AssertEquals(Expected := nExpectedState,
             Actual := nActualState,
             Message := 'State is not correct');	 
TEST_FINISHED();

TEST('Transition S3>S1_2');
fbDS402.eState := E_DS402State.S3_SwitchedOn;
fbDS402.stControl := GetQuickStopCommand();
fbDS402.stControl.b1_EnableVoltage := TRUE;
fbDS402();

nExpectedState := E_DS402State.S1_SwitchOnDisabled;
nActualState := fbDS402.eState;

AssertEquals(Expected := nExpectedState,
             Actual := nActualState,
             Message := 'State is not correct');	 
TEST_FINISHED();

TEST('Transition S3>S2');
fbDS402.eState := E_DS402State.S3_SwitchedOn;
fbDS402.stControl := GetShotdownCommand();
fbDS402();

nExpectedState := E_DS402State.S2_ReadyToSwitchOn;
nActualState := fbDS402.eState;

AssertEquals(Expected := nExpectedState,
             Actual := nActualState,
             Message := 'State is not correct');	 
TEST_FINISHED();

TEST('Transition S3>S4');
fbDS402.eState := E_DS402State.S3_SwitchedOn;
fbDS402.stControl := GetEnableCommand();
fbDS402();

nExpectedState := E_DS402State.S4_OperationEnabled;
nActualState := fbDS402.eState;

AssertEquals(Expected := nExpectedState,
             Actual := nActualState,
             Message := 'State is not correct');	 
TEST_FINISHED();
END_METHOD

METHOD TestState_S4 : BOOL
VAR
	fbDS402 			: FB_DS402FSM;
	stExpectedStatus 	: ST_DS402_6041h_StatusWord; 
	nMask 				: WORD;
	nResult 			: WORD;
	bResult 			: BOOL;
	nActualState		: INT;
	nExpectedState		: INT;
END_VAR
TEST('Set State S4');
fbDS402.eState := E_DS402State.S4_OperationEnabled;
fbDS402();

stExpectedStatus.b0_ReadyToSwitchOn 		:= TRUE;
stExpectedStatus.b1_SwitchedOn 				:= TRUE;
stExpectedStatus.b2_OperationEnabled		:= TRUE;
stExpectedStatus.b3_Fault					:= FALSE;
stExpectedStatus.b5_QuickStop 				:= TRUE; 
stExpectedStatus.b6_SwitchOnDisabled 		:= FALSE;

MEMCPY(ADR(nMask), ADR(stExpectedStatus), 2);
nResult := (2#01101111 AND fbDS402.nStatus);

AssertEquals(Expected := nMask,
             Actual := nResult,
             Message := 'Value is not correct');	 
TEST_FINISHED();

TEST('Transition S4>S6');
fbDS402.eState := E_DS402State.S4_OperationEnabled;
fbDS402.bError := TRUE;
fbDS402();
fbDS402.bError := FALSE;

nExpectedState := E_DS402State.S6_FaultReactionActive;
nActualState := fbDS402.eState;

AssertEquals(Expected := nExpectedState,
             Actual := nActualState,
             Message := 'State is not correct');	 
TEST_FINISHED();

TEST('Transition S4>S1');
fbDS402.eState := E_DS402State.S4_OperationEnabled;
fbDS402.stControl := GetDisableVoltageCommand();
fbDS402();

nExpectedState := E_DS402State.S1_SwitchOnDisabled;
nActualState := fbDS402.eState;

AssertEquals(Expected := nExpectedState,
             Actual := nActualState,
             Message := 'State is not correct');	 
TEST_FINISHED();

TEST('Transition S4>S2');
fbDS402.eState := E_DS402State.S4_OperationEnabled;
fbDS402.stControl := GetShotdownCommand();
fbDS402();

nExpectedState := E_DS402State.S2_ReadyToSwitchOn;
nActualState := fbDS402.eState;

AssertEquals(Expected := nExpectedState,
             Actual := nActualState,
             Message := 'State is not correct');	 
TEST_FINISHED();

TEST('Transition S4>S3');
fbDS402.eState := E_DS402State.S4_OperationEnabled;
fbDS402.stControl := GetDisableCommand();
fbDS402();

nExpectedState := E_DS402State.S3_SwitchedOn;
nActualState := fbDS402.eState;

AssertEquals(Expected := nExpectedState,
             Actual := nActualState,
             Message := 'State is not correct');	 
TEST_FINISHED();

TEST('Transition S4>S7');
fbDS402.eState := E_DS402State.S4_OperationEnabled;
fbDS402.stControl := GetQuickStopCommand();
fbDS402.stControl.b1_EnableVoltage := TRUE;
fbDS402();

nExpectedState := E_DS402State.S7_QuickStopActive;
nActualState := fbDS402.eState;

AssertEquals(Expected := nExpectedState,
             Actual := nActualState,
             Message := 'State is not correct');	 
TEST_FINISHED();
END_METHOD

METHOD TestState_S5 : BOOL
VAR
	fbDS402 			: FB_DS402FSM;
	stExpectedStatus 	: ST_DS402_6041h_StatusWord; 
	nMask 				: WORD;
	nResult 			: WORD;
	bResult 			: BOOL;
	nActualState		: INT;
	nExpectedState		: INT;
END_VAR
TEST('Set State S5');
fbDS402.eState := E_DS402State.S5_Fault;
fbDS402();

stExpectedStatus.b0_ReadyToSwitchOn 		:= FALSE;
stExpectedStatus.b1_SwitchedOn 				:= FALSE;
stExpectedStatus.b2_OperationEnabled		:= FALSE;
stExpectedStatus.b3_Fault					:= TRUE;
stExpectedStatus.b6_SwitchOnDisabled 		:= FALSE;

MEMCPY(ADR(nMask), ADR(stExpectedStatus), 2);
nResult := (2#01001111 AND fbDS402.nStatus);

AssertEquals(Expected := nMask,
             Actual := nResult,
             Message := 'Value is not correct');	 
TEST_FINISHED();

TEST('Transition S5>S1');
fbDS402.eState := E_DS402State.S5_Fault;
fbDS402.stControl.b7_FaultReset := TRUE;
fbDS402();
fbDS402.stControl.b7_FaultReset := FALSE;

nExpectedState := E_DS402State.S1_SwitchOnDisabled;
nActualState := fbDS402.eState;

AssertEquals(Expected := nExpectedState,
             Actual := nActualState,
             Message := 'State is not correct');	 
TEST_FINISHED();
END_METHOD

METHOD TestState_S6 : BOOL
VAR
	fbDS402 			: FB_DS402FSM;
	stExpectedStatus 	: ST_DS402_6041h_StatusWord; 
	nMask 				: WORD;
	nResult 			: WORD;
	bResult 			: BOOL;
	nActualState		: INT;
	nExpectedState		: INT;
END_VAR
TEST('Set State S6');
fbDS402.eState := E_DS402State.S6_FaultReactionActive;
fbDS402();

stExpectedStatus.b0_ReadyToSwitchOn 		:= TRUE;
stExpectedStatus.b1_SwitchedOn 				:= TRUE;
stExpectedStatus.b2_OperationEnabled		:= TRUE;
stExpectedStatus.b3_Fault					:= TRUE;
stExpectedStatus.b6_SwitchOnDisabled 		:= FALSE;

MEMCPY(ADR(nMask), ADR(stExpectedStatus), 2);
nResult := (2#01001111 AND fbDS402.nStatus);

AssertEquals(Expected := nMask,
             Actual := nResult,
             Message := 'Value is not correct');	 
TEST_FINISHED();

TEST('Transition S6>S5');
fbDS402.eState := E_DS402State.S6_FaultReactionActive;
fbDS402();

nExpectedState := E_DS402State.S5_Fault;
nActualState := fbDS402.eState;

AssertEquals(Expected := nExpectedState,
             Actual := nActualState,
             Message := 'State is not correct');	 
TEST_FINISHED();
END_METHOD

METHOD TestState_S7 : BOOL
VAR
	fbDS402 			: FB_DS402FSM;
	stExpectedStatus 	: ST_DS402_6041h_StatusWord; 
	nMask 				: WORD;
	nResult 			: WORD;
	bResult 			: BOOL;
	nActualState		: INT;
	nExpectedState		: INT;
END_VAR
TEST('Set State S7');
fbDS402.eState := E_DS402State.S7_QuickStopActive;
fbDS402();

stExpectedStatus.b0_ReadyToSwitchOn 		:= TRUE;
stExpectedStatus.b1_SwitchedOn 				:= TRUE;
stExpectedStatus.b2_OperationEnabled		:= TRUE;
stExpectedStatus.b3_Fault					:= FALSE;
stExpectedStatus.b5_QuickStop				:= FALSE;
stExpectedStatus.b6_SwitchOnDisabled 		:= FALSE;

MEMCPY(ADR(nMask), ADR(stExpectedStatus), 2);
nResult := (2#01101111 AND fbDS402.nStatus);

AssertEquals(Expected := nMask,
             Actual := nResult,
             Message := 'Value is not correct');	 
TEST_FINISHED();

TEST('Transition S7>S1');
fbDS402.eState := E_DS402State.S7_QuickStopActive;
fbDS402.stControl := GetDisableVoltageCommand();
fbDS402();

nExpectedState := E_DS402State.S1_SwitchOnDisabled;
nActualState := fbDS402.eState;

AssertEquals(Expected := nExpectedState,
             Actual := nActualState,
             Message := 'State is not correct');	 
TEST_FINISHED();

TEST('Transition S7>S4');
fbDS402.eState := E_DS402State.S7_QuickStopActive;
fbDS402.stControl := GetEnableCommand();
fbDS402();

nExpectedState := E_DS402State.S4_OperationEnabled;
nActualState := fbDS402.eState;

AssertEquals(Expected := nExpectedState,
             Actual := nActualState,
             Message := 'State is not correct');	 
TEST_FINISHED();
END_METHOD

END_FUNCTION_BLOCK

// Tests/Drives/FB_Encoder_Test
FUNCTION_BLOCK FB_Encoder_Test EXTENDS FB_TestSuite
VAR	
	stConfig 			: ST_EncoderConfig;
END_VAR

TestCase_Encoder('Absolute 1', 0, 0, LREAL_TO_DINT(0*1E4), stConfig);
TestCase_Encoder('Absolute 2', 100, 100, LREAL_TO_DINT(100*1E4), stConfig);
TestCase_Encoder('Absolute 3', -100, -100, LREAL_TO_DINT(-100*1E4), stConfig);

stConfig.fInputFactor := -1;
TestCase_Encoder('Absolute with Factor 1', 0, 0, LREAL_TO_DINT(0*1E4), stConfig);
TestCase_Encoder('Absolute with Factor 2', 100, -100, LREAL_TO_DINT(-100*1E4), stConfig);
TestCase_Encoder('Absolute with Factor 3', -100, 100, LREAL_TO_DINT(100*1E4), stConfig);

stConfig.fInputFactor := 1;
stConfig.bInvertIncrementValue := TRUE;
TestCase_Encoder('Absolute with Invert 1', 0, 0, LREAL_TO_DINT(0*1E4), stConfig);
TestCase_Encoder('Absolute with Invert 2', 100, 100, LREAL_TO_DINT(-100*1E4), stConfig);
TestCase_Encoder('Absolute with Invert 3', -100, -100, LREAL_TO_DINT(100*1E4), stConfig);

stConfig.fModulo := 360;
stConfig.bInvertIncrementValue := FALSE;
TestCase_Encoder('Modulo 1', 0, 0, LREAL_TO_DINT(0*1E4), stConfig);
TestCase_Encoder('Modulo 2', 360, 0, LREAL_TO_DINT(0*1E4), stConfig);
TestCase_Encoder('Modulo 3', 350, 350, LREAL_TO_DINT(350*1E4), stConfig);
TestCase_Encoder('Modulo 4', -350, -350, LREAL_TO_DINT(-350*1E4), stConfig);
TestCase_Encoder('Modulo 5', -360, 0, LREAL_TO_DINT(0*1E4), stConfig);

stConfig.fModulo := 0;
stConfig.bInvertIncrementValue := FALSE;
stConfig.bIsIntegral := TRUE;
TestCase_Encoder('Integrate 1', 0, 0, 0, stConfig);
TestCase_Encoder('Integrate 2', 100, 1, LREAL_TO_DINT(1*1E4), stConfig);
TestCase_Encoder('Integrate 3', -100, -1, LREAL_TO_DINT(-1*1E4), stConfig);

METHOD TestCase_Encoder
VAR_INPUT
	sName 					: T_MaxString;
	fInput					: REAL;
	fExpected				: LREAL;
	nExpected				: DINT;
	stConfig				: ST_EncoderConfig;
END_VAR

VAR	
	fbEncoder 				: FB_Encoder;
	nCycleCount 			: INT;
	fActual					: LREAL;	
	nActual					: DINT;	
	bValid 					: BOOL;
	fTolerance 				: REAL := 1E-6;
END_VAR
TEST(sName);

fbEncoder.stConfig := stConfig;
fbEncoder.fInput := fInput;

(*	Call FB to test	*)
FOR nCycleCount := 0 TO 9 DO
   fbEncoder();
END_FOR

(*	Evaluation of results	*)
nActual := fbEncoder.nPosition;
fActual := fbEncoder.fPosition;

AssertEquals(Expected := nExpected,
             Actual := nActual,
             Message := 'nPosition is not correct');

bValid := ABS(fExpected - fActual) < fTolerance;			 
	
AssertTrue(bValid, 'fPosition is not correct');

TEST_FINISHED();
END_METHOD

END_FUNCTION_BLOCK

// Tests/Drives/FB_SimMovidriveFSM_Test
FUNCTION_BLOCK FB_SimMovidriveFSM_Test EXTENDS TcUnit.FB_TestSuite

// TestState(sTestInfo, bControllerInhibit, bRapidStop,	bStop,	bHoldControl, eInitState, eExpectedState)	

// ControllerInhibit
TestState('ControllerInhibit, no transition', TRUE, FALSE, FALSE, FALSE, E_SimMovitracState.ControllerInhibit, E_SimMovitracState.ControllerInhibit);
TestState('ControllerInhibit -> RapidStop', FALSE, FALSE, FALSE, FALSE, E_SimMovitracState.ControllerInhibit, E_SimMovitracState.RapidStop);

//  RapidStop 
TestState('RapidStop, no transition', FALSE, FALSE, FALSE, FALSE, E_SimMovitracState.RapidStop, E_SimMovitracState.RapidStop);
TestState('RapidStop -> ControllerInhibit', TRUE, FALSE, FALSE, FALSE, E_SimMovitracState.RapidStop, E_SimMovitracState.ControllerInhibit);
TestState('RapidStop -> Halt', FALSE, TRUE, FALSE, FALSE, E_SimMovitracState.RapidStop, E_SimMovitracState.Halt);

// Halt
TestState('Halt, no transition', FALSE, TRUE, FALSE, FALSE, E_SimMovitracState.Halt, E_SimMovitracState.Halt);
TestState('Halt -> ControllerInhibit', TRUE, FALSE, FALSE, FALSE, E_SimMovitracState.Halt, E_SimMovitracState.ControllerInhibit);
TestState('Halt -> RapidStop', FALSE, FALSE, FALSE, FALSE, E_SimMovitracState.Halt, E_SimMovitracState.RapidStop);
TestState('Halt -> HoldControl', FALSE, TRUE, TRUE, TRUE, E_SimMovitracState.Halt, E_SimMovitracState.HoldControl);
TestState('Halt -> Enable', FALSE, TRUE, TRUE, FALSE, E_SimMovitracState.Halt, E_SimMovitracState.Enable);

// Enable
TestState('Enable, no transition', FALSE, TRUE, TRUE, FALSE, E_SimMovitracState.Enable, E_SimMovitracState.Enable);
TestState('Enable -> ControllerInhibit', TRUE, FALSE, FALSE, FALSE, E_SimMovitracState.Enable, E_SimMovitracState.ControllerInhibit);
TestState('Enable -> RapidStop', FALSE, FALSE, FALSE, FALSE, E_SimMovitracState.Enable, E_SimMovitracState.RapidStop);
TestState('Enable -> Halt', FALSE, TRUE, FALSE, FALSE, E_SimMovitracState.Enable, E_SimMovitracState.Halt);
TestState('Enable -> HoldControl', FALSE, TRUE, TRUE, TRUE, E_SimMovitracState.Enable, E_SimMovitracState.HoldControl);

// HoldControl
TestState('HoldControl, no transition', FALSE, TRUE, TRUE, TRUE, E_SimMovitracState.HoldControl, E_SimMovitracState.HoldControl);
TestState('HoldControl -> ControllerInhibit', TRUE, FALSE, FALSE, FALSE, E_SimMovitracState.HoldControl, E_SimMovitracState.ControllerInhibit);
TestState('HoldControl -> RapidStop', FALSE, FALSE, FALSE, FALSE, E_SimMovitracState.HoldControl, E_SimMovitracState.RapidStop);
TestState('HoldControl -> Halt', FALSE, TRUE, FALSE, FALSE, E_SimMovitracState.HoldControl, E_SimMovitracState.Halt);
TestState('HoldControl -> Enable', FALSE, TRUE, TRUE, FALSE, E_SimMovitracState.HoldControl, E_SimMovitracState.Enable);

METHOD TestState : BOOL
VAR_INPUT
	sTestInfo			: T_MaxString;
	bControllerInhibit	: BOOL;
	bRapidStop			: BOOL;
	bStop				: BOOL;
	bHoldControl		: BOOL;
	eInitState			: E_SimMovitracState;	
	eExpectedState		: E_SimMovitracState;	
END_VAR

VAR
		fbMovidriveStateMachine		: FB_SimMovitracFSM;
END_VAR
TEST(sTestInfo);

fbMovidriveStateMachine.bControllerInhibit := bControllerInhibit;
fbMovidriveStateMachine.bRapidStop := bRapidStop;
fbMovidriveStateMachine.bStop := bStop;
fbMovidriveStateMachine.bHoldControl := bHoldControl;

fbMovidriveStateMachine.nState := eInitState;

fbMovidriveStateMachine();

AssertEquals(Expected := eExpectedState,
             Actual := fbMovidriveStateMachine.eState,
             Message := 'State is not correct');
	 
TEST_FINISHED();
END_METHOD

END_FUNCTION_BLOCK

// Tests/Drives/FB_SimMovidrivePDO12_Test
FUNCTION_BLOCK FB_SimMovidrivePDO12_Test EXTENDS TcUnit.FB_TestSuite
VAR_INPUT
END_VAR
VAR_OUTPUT
END_VAR
VAR
END_VAR

Test_GetControlMode();
Test_GetControlData();
Test_GetControlDataSWAP();
Test_SetStatusData();
Test_SetStatusDataSWAP();

METHOD Test_AssignProcessData : REFERENCE TO FB_Test
VAR
	fbStarter 				: FB_Starter;
	nControlData 			: WORD;
	nStatusData				: WORD;
	
	nExpectedStatusData		: WORD;
	
	nActualControlData 		: WORD;
	nActualStatusData		: WORD;
	stActualControlData 	: ST_StarterControlData;
	stActualStatusData		: ST_StarterStatusData;
END_VAR
TEST('Assign Process data');

nControlData := 255;
nStatusData := 0;

fbStarter.AssignProcessData(nControlData, nStatusData);
fbStarter();

stActualControlData := fbStarter.stControlData;
stActualStatusData := fbStarter.stStatusData;

MEMCPY(ADR(nActualControlData), ADR(stActualControlData), 2);
MEMCPY(ADR(nActualStatusData), ADR(stActualStatusData), 2);

AssertEquals(Expected := nControlData,
             Actual := nActualControlData,
             Message := 'nControlData is not correct');	
		
nExpectedStatusData := 1;
	 
AssertEquals(Expected := nExpectedStatusData,
             Actual := nStatusData,
             Message := 'nStatusData is not correct');	

TEST_FINISHED();
END_METHOD

METHOD Test_GetControlData : BOOL
VAR
	stDataBus 		: ST_SimMovidriveControlData;
	stControl 		: ST_SimMovidriveControlData;
	stExpected 		: ST_SimMovidriveControlData;
	fbMoviPos_PD12 	: FB_SimMovidrivePDO12;
	
	nControlWord	: WORD;
	nControlWordExpected	: WORD;
END_VAR
TEST('Get Control Data');

stDataBus.bControllerInhibit := TRUE;
stDataBus.nTargetPosition := 100;
stDataBus.nVelocity := 200;
stDataBus.nAcceleration := 300;
stDataBus.nDeceleration := 400;

stExpected := stDataBus;
MEMCPY(ADR(nControlWordExpected), ADR(stExpected), 2);

fbMoviPos_PD12.GetControlData(stControl, ADR(stDataBus), FALSE);
MEMCPY(ADR(nControlWord), ADR(stControl), 2);

AssertEquals(Expected := nControlWordExpected,
             Actual := nControlWord,
             Message := 'nControlWord is not equal');
			 
AssertEquals(Expected := stExpected.nTargetPosition,
             Actual := stControl.nTargetPosition,
             Message := 'nTargetPosition word is not equal');
			 
AssertEquals(Expected := stExpected.nVelocity,
             Actual := stControl.nVelocity,
             Message := 'nVelocity word is not equal');	
			 
AssertEquals(Expected := stExpected.nAcceleration,
             Actual := stControl.nAcceleration,
             Message := 'nAcceleration word is not equal');	

AssertEquals(Expected := stExpected.nDeceleration,
             Actual := stControl.nDeceleration,
             Message := 'nAcceleration word is not equal');		 
		
TEST_FINISHED();
END_METHOD

METHOD Test_GetControlDataSWAP : BOOL
VAR
	stDataBus 				: ST_SimMovidriveControlData;
	stControl 				: ST_SimMovidriveControlData;
	stExpected 				: ST_SimMovidriveControlData;
	fbMoviPos_PD12 			: FB_SimMovidrivePDO12;
	                		
	nControlWord			: WORD;
	nControlWordExpected	: WORD;	
	nBusControlWord			: WORD;
END_VAR
TEST('Get Control Data SWAP');

nControlWordExpected := 15;
MEMCPY(ADR(stExpected), ADR(nControlWordExpected), 2);
stExpected.nTargetPosition := 100;
stExpected.nVelocity := 200;
stExpected.nAcceleration := 300;
stExpected.nDeceleration := 400;

stDataBus := stExpected ;
MEMCPY(ADR(nBusControlWord), ADR(stDataBus), 2);
nBusControlWord := HOST_TO_BE16(nBusControlWord);
MEMCPY(ADR(stDataBus), ADR(nBusControlWord), 2);

stDataBus.nTargetPosition := DWORD_TO_DINT(HOST_TO_BE32(DINT_TO_DWORD(stDataBus.nTargetPosition)));
stDataBus.nVelocity := HOST_TO_BE16(stDataBus.nVelocity);
stDataBus.nAcceleration := HOST_TO_BE16(stDataBus.nAcceleration);
stDataBus.nDeceleration := HOST_TO_BE16(stDataBus.nDeceleration);

fbMoviPos_PD12.GetControlData(stControl, ADR(stDataBus), TRUE);
MEMCPY(ADR(nControlWord), ADR(stControl), 2);

AssertEquals(Expected := nControlWordExpected,
             Actual := nControlWord,
             Message := 'nControlWord is not equal');
			 
AssertEquals(Expected := stExpected.nTargetPosition,
             Actual := stControl.nTargetPosition,
             Message := 'nTargetPosition word is not equal');
			 
AssertEquals(Expected := stExpected.nVelocity,
             Actual := stControl.nVelocity,
             Message := 'nVelocity word is not equal');	
			 
AssertEquals(Expected := stExpected.nAcceleration,
             Actual := stControl.nAcceleration,
             Message := 'nAcceleration word is not equal');	

AssertEquals(Expected := stExpected.nDeceleration,
             Actual := stControl.nDeceleration,
             Message := 'nAcceleration word is not equal');		 
		
TEST_FINISHED();
END_METHOD

METHOD Test_GetControlMode : REFERENCE TO FB_Test
VAR
	stControl 		: ST_SimMovidriveControlData;
	fbMoviPos_PD12 	: FB_SimMovidrivePDO12;
	bExpected		: BOOL;
	bResult			: BOOL;
END_VAR
TEST('Get Control Mode');

stControl.bModeLow := FALSE;
stControl.bModeHigh := FALSE;
bResult := fbMoviPos_PD12.GetControlMode(stControl) = E_SimMovidriveMode.Idle;
AssertTrue(bResult, 'Expected Idle Mode');


stControl.bModeLow := TRUE;
stControl.bModeHigh := FALSE;
bResult := fbMoviPos_PD12.GetControlMode(stControl) = E_SimMovidriveMode.Jog;
AssertTrue(bResult, 'Expected Jog Mode');

stControl.bModeLow := FALSE;
stControl.bModeHigh := TRUE;
bResult := fbMoviPos_PD12.GetControlMode(stControl) = E_SimMovidriveMode.Ref;
AssertTrue(bResult, 'Expected Ref Mode');

stControl.bModeLow := TRUE;
stControl.bModeHigh := TRUE;
bResult := fbMoviPos_PD12.GetControlMode(stControl) = E_SimMovidriveMode.Auto;
AssertTrue(bResult, 'Expected Auto Mode');

TEST_FINISHED();
END_METHOD

METHOD Test_SetStatusData : BOOL
VAR
	stControl 				: ST_SimMovidriveStatusData;
	stBuffer				: ST_SimMovidriveStatusData;
	fbMoviPos_PD12 			: FB_SimMovidrivePDO12;	                		
	nControlStatusByte		: BYTE;
	nActualStatusByte		: BYTE;
	nStatusWordSwap			: WORD;
END_VAR
TEST('Set Status Data');

nControlStatusByte := 124;
MEMCPY(ADR(stControl), ADR(nControlStatusByte), 1);
stControl.nStatus := 164;
stControl.nActPosition := 100;
stControl.nActVelocity := 200;
stControl.nActCurrent := 300;
stControl.nActUnit := 400;

fbMoviPos_PD12.SetStatusData(stControl, ADR(stBuffer), FALSE);

MEMCPY(ADR(nActualStatusByte), ADR(stBuffer), 1);

AssertEquals(Expected := nControlStatusByte,
             Actual := nActualStatusByte,
             Message := 'nExpectedStatusByte is not equal');

AssertEquals(Expected := stControl.nStatus,
             Actual := stBuffer.nStatus,
             Message := 'nStatus word is not equal');	

AssertEquals(Expected := stControl.nActPosition,
             Actual := stBuffer.nActPosition,
             Message := 'nActPosition word is not equal'); 
			 
AssertEquals(Expected := stControl.nActVelocity,
             Actual := stBuffer.nActVelocity,
             Message := 'nActVelocity word is not equal');
			 
AssertEquals(Expected := stControl.nActCurrent,
             Actual := stBuffer.nActCurrent,
             Message := 'nActCurrent word is not equal');
			 
AssertEquals(Expected := stControl.nActUnit,
             Actual := stBuffer.nActUnit,
             Message := 'nActCurrent word is not equal');

TEST_FINISHED();
END_METHOD

METHOD Test_SetStatusDataSWAP : BOOL
VAR
	stControl 				: ST_SimMovidriveStatusData;
	stBuffer				: ST_SimMovidriveStatusData;
	fbMoviPos_PD12 			: FB_SimMovidrivePDO12;	                		
	nControlStatusByte		: BYTE;
	nActualStatusByte		: BYTE;
	nStatusWordSwap			: WORD;
END_VAR
TEST('Set Status Data SWAP');

nControlStatusByte := 124;
MEMCPY(ADR(stControl), ADR(nControlStatusByte), 1);
stControl.nStatus := 164;
stControl.nActPosition := 100;
stControl.nActVelocity := 200;
stControl.nActCurrent := 300;
stControl.nActUnit := 400;

fbMoviPos_PD12.SetStatusData(stControl, ADR(stBuffer), TRUE);

MEMCPY(ADR(nStatusWordSwap), ADR(stBuffer), 2);
nStatusWordSwap := HOST_TO_BE16(nStatusWordSwap);
MEMCPY(ADR(stBuffer), ADR(nStatusWordSwap), 2);
stBuffer.nActPosition := DWORD_TO_DINT(HOST_TO_BE32(DINT_TO_DWORD(stBuffer.nActPosition)));
stBuffer.nActVelocity := HOST_TO_BE16(stBuffer.nActVelocity);
stBuffer.nActCurrent := HOST_TO_BE16(stBuffer.nActCurrent);
stBuffer.nActUnit := HOST_TO_BE16(stBuffer.nActUnit);

MEMCPY(ADR(nActualStatusByte), ADR(stBuffer), 1);

AssertEquals(Expected := nControlStatusByte,
             Actual := nActualStatusByte,
             Message := 'nExpectedStatusByte is not equal');

AssertEquals(Expected := stControl.nStatus,
             Actual := stBuffer.nStatus,
             Message := 'nStatus word is not equal');	

AssertEquals(Expected := stControl.nActPosition,
             Actual := stBuffer.nActPosition,
             Message := 'nActPosition word is not equal'); 
			 
AssertEquals(Expected := stControl.nActVelocity,
             Actual := stBuffer.nActVelocity,
             Message := 'nActVelocity word is not equal');
			 
AssertEquals(Expected := stControl.nActCurrent,
             Actual := stBuffer.nActCurrent,
             Message := 'nActCurrent word is not equal');
			 
AssertEquals(Expected := stControl.nActUnit,
             Actual := stBuffer.nActUnit,
             Message := 'nActUnit word is not equal');

TEST_FINISHED();
END_METHOD

END_FUNCTION_BLOCK

// Tests/Drives/FB_SimMovitrac_Test
FUNCTION_BLOCK FB_SimMovitrac_Test EXTENDS FB_TestSuite
VAR
	fbMovitrac : FB_SimMovitrac;
END_VAR

// No Movement
Test_Movitrac('No Movement, No STO', FALSE, FALSE, TRUE, TRUE, 1000, 0, FALSE, 10);
Test_Movitrac('No Movement, ControllerInhibit', TRUE, TRUE, TRUE, TRUE, 1000, 0, FALSE, 10);
Test_Movitrac('No Movement, No RapidStop', TRUE, FALSE, FALSE, TRUE, 1000, 0, FALSE, 10);
Test_Movitrac('No Movement, No Stop', TRUE, FALSE, TRUE, FALSE, 1000, 0, FALSE, 10);

// Movement
Test_Movitrac('Velocity postive', TRUE, FALSE, TRUE, TRUE, 1000, 1000, TRUE, 50);
Test_Movitrac('Velocity negative', TRUE, FALSE, TRUE, TRUE, -1000, -1000, TRUE, 50);
Test_Movitrac('Velocity 0', TRUE, FALSE, TRUE, TRUE, 0, 0, FALSE, 50);

// Stop
Test_Movitrac('Velocity to Stop', TRUE, FALSE, TRUE, TRUE, 1000, 1000, TRUE, 50);
Test_Movitrac('Stop', TRUE, FALSE, TRUE, FALSE, 0, 0, FALSE, 50);

// Rapid Stop
Test_Movitrac('Velocity to Rapid Stop', TRUE, FALSE, TRUE, TRUE, 1000, 1000, TRUE, 50);
Test_Movitrac('Rapid Stop', TRUE, FALSE, FALSE, TRUE, 0, 0, FALSE, 50);

// STO Stop
Test_Movitrac('Velocity to STO Stop', TRUE, FALSE, TRUE, TRUE, 1000, 1000, TRUE, 50);
Test_Movitrac('STO Stop', FALSE, FALSE, TRUE, TRUE, 0, 0, FALSE, 50);

METHOD Test_Movitrac
VAR
	nCycleCount : INT;
	bResultOutputStage : BOOL;
END_VAR
VAR_INPUT
	sTestInfo			: T_MaxString;
	bSto				: BOOL;
	bControllerInhibit	: BOOL;
	bRapidStop			: BOOL;
	bStop				: BOOL;
	nSetpointSpeed		: INT;	
	eExpectedSpeed		: INT;
	bExpectedOutputStage: BOOL;		
	bCycles				: INT;	
END_VAR
TEST(sTestInfo);

fbMovitrac.bSTO := bSTO;
fbMovitrac.stControlData.bControllerInhibit := bControllerInhibit;
fbMovitrac.stControlData.bRapidStop := bRapidStop;
fbMovitrac.stControlData.bStop := bStop;
fbMovitrac.stControlData.nSetpointSpeed := nSetpointSpeed; 

FOR nCycleCount := 0 TO bCycles DO
    fbMovitrac();
END_FOR

bResultOutputStage := fbMovitrac.stStatusData.bEnableOutputStage;

AssertEquals(Expected := eExpectedSpeed,
             Actual := fbMovitrac.stStatusData.nActSpeed,
             Message := 'Velocity/Speed is not correct');
			 
AssertEquals(Expected := bExpectedOutputStage,
             Actual := bResultOutputStage,
             Message := 'EnableOutputStage is not correct');

TEST_FINISHED();
END_METHOD

END_FUNCTION_BLOCK

// Tests/Drives/FB_SimMovitracB_Test
FUNCTION_BLOCK FB_SimMovitracB_Test EXTENDS FB_TestSuite
VAR
	fbMovitracB : FB_SimMovitracB;
END_VAR

// No Movement
TestCase_SimMovitracB('No Movement, No STO', FALSE, FALSE, TRUE, TRUE, 32767, 0, FALSE);
TestCase_SimMovitracB('No Movement, ControllerInhibit', TRUE, TRUE, TRUE, TRUE, 32767, 0, FALSE);
TestCase_SimMovitracB('No Movement, No RapidStop', TRUE, FALSE, FALSE, TRUE, 32767, 0, FALSE);
TestCase_SimMovitracB('No Movement, No Stop', TRUE, FALSE, TRUE, FALSE, 32767, 0, FALSE);

// Movement
TestCase_SimMovitracB('Velocity postive', TRUE, FALSE, TRUE, TRUE, 32767, 3000, TRUE);
TestCase_SimMovitracB('Velocity negative', TRUE, FALSE, TRUE, TRUE, -32767, -3000, TRUE);
TestCase_SimMovitracB('Velocity 0', TRUE, FALSE, TRUE, TRUE, 0, 0, FALSE);

// Stop
TestCase_SimMovitracB('Velocity to Stop', TRUE, FALSE, TRUE, TRUE, 32767, 3000, TRUE);
TestCase_SimMovitracB('Stop', TRUE, FALSE, TRUE, FALSE, 0, 0, FALSE);

// STO Stop
TestCase_SimMovitracB('Velocity to STO Stop', TRUE, FALSE, TRUE, TRUE, 32767, 3000, TRUE);
TestCase_SimMovitracB('STO Stop', FALSE, FALSE, TRUE, TRUE, 0, 0, FALSE);

// Rapid Stop
TestCase_SimMovitracB('Velocity to Rapid Stop', TRUE, FALSE, TRUE, TRUE, 32767, 3000, TRUE);
TestCase_SimMovitracB('Rapid Stop', TRUE, FALSE, FALSE, TRUE, 0, 0, FALSE);

METHOD TestCase_SimMovitracB
VAR
	nCycleCount : INT;
	bResultOutputStage : BOOL;
END_VAR
VAR_INPUT
	sTestInfo			: T_MaxString;
	bSto				: BOOL;
	bControllerInhibit	: BOOL;
	bRapidStop			: BOOL;
	bStop				: BOOL;
	nSetpointSpeed		: INT;	
	eExpectedSpeed		: REAL;
	bExpectedOutputStage: BOOL;		
END_VAR
TEST(sTestInfo);

fbMovitracB.bSTO := bSTO;
fbMovitracB.stControlData.bControllerInhibit := bControllerInhibit;
fbMovitracB.stControlData.bRapidStop := bRapidStop;
fbMovitracB.stControlData.bStop := bStop;
fbMovitracB.stControlData.nSetpointSpeed := nSetpointSpeed; 

fbMovitracB();

bResultOutputStage := fbMovitracB.stStatusData.bEnableOutputStage;

AssertEquals(Expected := eExpectedSpeed,
             Actual := fbMovitracB.fVelocity,
             Message := 'Velocity/Speed is not correct');
			 
AssertEquals(Expected := bExpectedOutputStage,
             Actual := bResultOutputStage,
             Message := 'EnableOutputStage is not correct');

TEST_FINISHED();
END_METHOD

END_FUNCTION_BLOCK

// Tests/Drives/FB_SimMovitracLTEB_Test
FUNCTION_BLOCK FB_SimMovitracLTEB_Test EXTENDS FB_TestSuite
VAR
	fbMovitracLTE : FB_SimMovitracLTEB;
	nExpectedByte : BYTE;
	nResultByte : BYTE;
	fExpectedReal : REAL;
	fResultReal : REAL;
	bExpectedBool : BOOL;
	bResultBool : BOOL;
END_VAR

Test_DriveNotReady();
Test_DriveReady();
Test_DriveRunningFwd();
Test_DriveRunningBwd();

METHOD Test_DriveNotReady
VAR_INPUT
END_VAR
TEST('Drive is not ready');
nExpectedByte := 0; 
bExpectedBool := FALSE;
fbMovitracLTE.bEnable := FALSE;
fbMovitracLTE.bSTO := FALSE;
fbMovitracLTE();
nResultByte := fbMovitracLTE.GetControl();
bResultBool := fbMovitracLTE.bReady;
AssertEquals(Expected := nExpectedByte,
             Actual := nResultByte,
             Message := 'Value is not correct');

AssertEquals(Expected := bExpectedBool, 
			 Actual := bResultBool,
			 Message := 'Status is not correct');	
TEST_FINISHED();
END_METHOD

METHOD Test_DriveReady
VAR_INPUT
END_VAR
TEST('Drive is ready');
nExpectedByte := 0; 
bExpectedBool := TRUE;
fbMovitracLTE.bEnable := FALSE;
fbMovitracLTE.bSTO := TRUE;
fbMovitracLTE();
nResultByte := fbMovitracLTE.GetControl();
bResultBool := fbMovitracLTE.bReady;

AssertEquals(Expected := nExpectedByte,
             Actual := nResultByte,
             Message := 'Value is not correct');

AssertEquals(Expected := bExpectedBool,
			 Actual := bResultBool,
			 Message := 'Status is not correct');	
TEST_FINISHED();
END_METHOD

METHOD Test_DriveRunningBwd
VAR_INPUT
END_VAR
TEST('Drive is running backward with 0 speed');
fbMovitracLTE.bSTO := TRUE;
fbMovitracLTE.bReverse := TRUE;
fExpectedReal := 0;
bExpectedBool := TRUE;
fbMovitracLTE.bEnable := TRUE;
fbMovitracLTE.nTargetSpeed := 0;
fbMovitracLTE.SetStatus(1);
fbMovitracLTE();
fResultReal := fbMovitracLTE.GetLinkControlData();
bResultBool := fbMovitracLTE.bRunning;

AssertEquals(Expected := fExpectedReal,
             Actual := fResultReal,
             Message := 'DataOut is not correct');	
			 
AssertEquals(Expected := bExpectedBool,
             Actual := bResultBool,
             Message := 'Status is not correct');	
			 
TEST_FINISHED();
//######################################################
TEST('Feedback of Drive running backward with 0 speed');
fbMovitracLTE.bSTO := TRUE;
fbMovitracLTE.bReverse := TRUE;
fExpectedReal := 0;
bExpectedBool := TRUE;
fbMovitracLTE.bEnable := TRUE;
fbMovitracLTE.nTargetSpeed := 0;
fbMovitracLTE.SetLinkStatusData(fExpectedReal);
fbMovitracLTE.SetStatus(1);
fbMovitracLTE();
fResultReal := fbMovitracLTE.fActualSpeed;
bResultBool := fbMovitracLTE.bRunning;

AssertEquals(Expected := fExpectedReal,
             Actual := fResultReal,
             Message := 'DataIn is not correct');	
			 
AssertEquals(Expected := bExpectedBool,
             Actual := bResultBool,
             Message := 'Status is not correct');	
			 
TEST_FINISHED();
//######################################################
TEST('Drive is running backward at max speed');
fbMovitracLTE.bSTO := TRUE;
fbMovitracLTE.bReverse := TRUE;
fExpectedReal := -3000.0;
bExpectedBool := TRUE;
fbMovitracLTE.bEnable := TRUE;
fbMovitracLTE.nTargetSpeed := 65535;
fbMovitracLTE.SetStatus(1);
fbMovitracLTE();
fResultReal := fbMovitracLTE.GetLinkControlData();
bResultBool := fbMovitracLTE.bRunning;

AssertEquals(Expected := fExpectedReal,
             Actual := fResultReal,
             Message := 'DataOut is not correct');	
			 
AssertEquals(Expected := bExpectedBool,
             Actual := bResultBool,
             Message := 'Status is not correct');	
			 
TEST_FINISHED();
//###################################################
TEST('Feedback of Drive running backward at max speed');
fbMovitracLTE.bSTO := TRUE;
fbMovitracLTE.bReverse := TRUE;
fExpectedReal := 0;
bExpectedBool := TRUE;
fbMovitracLTE.bEnable := TRUE;
fbMovitracLTE.nTargetSpeed := 0;
fbMovitracLTE.SetStatus(1);
fbMovitracLTE.SetLinkStatusData(fExpectedReal);
fbMovitracLTE();
fResultReal := fbMovitracLTE.fActualSpeed;
bResultBool := fbMovitracLTE.bRunning;

AssertEquals(Expected := fExpectedReal,
             Actual := fResultReal,
             Message := 'DataIn is not correct');	
			 
AssertEquals(Expected := bExpectedBool,
             Actual := bResultBool,
             Message := 'Status is not correct');	
			 
TEST_FINISHED();
END_METHOD

METHOD Test_DriveRunningFwd
VAR_INPUT
END_VAR
TEST('Drive is running forward at 0');
fExpectedReal := 0;
bExpectedBool := TRUE;
fbMovitracLTE.bSTO := TRUE;
fbMovitracLTE.nTargetSpeed := 0;
fbMovitracLTE.bEnable := TRUE;
fbMovitracLTE.SetStatus(1);
fbMovitracLTE();
fResultReal := fbMovitracLTE.GetLinkControlData();
bResultBool := fbMovitracLTE.bRunning;

AssertEquals(Expected := fExpectedReal,
             Actual := fResultReal,
             Message := 'DataOut is not correct');	

AssertEquals(Expected := bExpectedBool, 
			 Actual := bResultBool,
			 Message := 'Status is not correct');
TEST_FINISHED();
//#################################################################
TEST('Feedback of drive running forward at 0');
fExpectedReal := 0;
bExpectedBool := TRUE;
fbMovitracLTE.bSTO := TRUE;
fbMovitracLTE.nTargetSpeed := 0;
fbMovitracLTE.bEnable := TRUE;
fbMovitracLTE.SetStatus(1);
fbMovitracLTE.SetLinkStatusData(fExpectedReal);
fbMovitracLTE();
fResultReal := fbMovitracLTE.fActualSpeed;
bResultBool := fbMovitracLTE.bRunning;

AssertEquals(Expected := fExpectedReal,
             Actual := fResultReal,
             Message := 'DataIn is not correct');	

AssertEquals(Expected := bExpectedBool, 
			 Actual := bResultBool,
			 Message := 'Status is not correct');
TEST_FINISHED();
//###################################################################
TEST('Drive is running forward at max speed');
fExpectedReal := 3000;
bExpectedBool := TRUE;
fbMovitracLTE.bSTO := TRUE;
fbMovitracLTE.nTargetSpeed := 65535;
fbMovitracLTE.bEnable := TRUE;
fbMovitracLTE.SetStatus(1);
fbMovitracLTE();
fResultReal := fbMovitracLTE.GetLinkControlData();
bResultBool := fbMovitracLTE.bRunning;

AssertEquals(Expected := fExpectedReal,
             Actual := fResultReal,
             Message := 'DataOut is not correct');	

AssertEquals(Expected := bExpectedBool, 
			 Actual := bResultBool,
			 Message := 'Status is not correct');
TEST_FINISHED();
//###################################################################
TEST('Feedback of drive running forward at max speed');
fExpectedReal := 3000;
bExpectedBool := TRUE;
fbMovitracLTE.bSTO := TRUE;
fbMovitracLTE.nTargetSpeed := 65535;
fbMovitracLTE.bEnable := TRUE;
fbMovitracLTE.SetStatus(1);
fbMovitracLTE.SetLinkStatusData(fExpectedReal);
fbMovitracLTE();
fResultReal := fbMovitracLTE.fActualSpeed;
bResultBool := fbMovitracLTE.bRunning;

AssertEquals(Expected := fExpectedReal,
             Actual := fResultReal,
             Message := 'DataIn is not correct');	

AssertEquals(Expected := bExpectedBool, 
			 Actual := bResultBool,
			 Message := 'Status is not correct');
TEST_FINISHED();
END_METHOD

END_FUNCTION_BLOCK

// Tests/Drives/FB_Starter_Test
FUNCTION_BLOCK FB_Starter_Test EXTENDS FB_TestSuite
VAR
	fbStarter : FB_Starter;
	
	fExpectedReal 		: REAL;
	fResultReal 		: REAL;
	bExpectedBool 		: BOOL;
	bResultBool 		: BOOL;
	fExpectedDataOut 	: REAL;
END_VAR

Test_GetControlData();
Test_GetControlDataSWAP();
Test_SetStatusData();
Test_SetStatusDataSWAP();

//Test_DriveNoMovement();
//Test_DriveRunningCw();
//Test_DriveRunningCcw();
//Test_AssignProcessData();

METHOD Test_AssignProcessData : REFERENCE TO FB_Test
VAR
	fbStarter 				: FB_Starter;
	nControlData 			: WORD;
	nStatusData				: WORD;
	
	nExpectedStatusData		: WORD;
	
	nActualControlData 		: WORD;
	nActualStatusData		: WORD;
	stActualControlData 	: ST_StarterControlData;
	stActualStatusData		: ST_StarterStatusData;
END_VAR
TEST('Assign Process data');

nControlData := 255;
nStatusData := 0;

fbStarter.AssignProcessData(nControlData, nStatusData);
fbStarter();

stActualControlData := fbStarter.stControlData;
stActualStatusData := fbStarter.stStatusData;

MEMCPY(ADR(nActualControlData), ADR(stActualControlData), 2);
MEMCPY(ADR(nActualStatusData), ADR(stActualStatusData), 2);

AssertEquals(Expected := nControlData,
             Actual := nActualControlData,
             Message := 'nControlData is not correct');	
		
nExpectedStatusData := 1;
	 
AssertEquals(Expected := nExpectedStatusData,
             Actual := nStatusData,
             Message := 'nStatusData is not correct');	

TEST_FINISHED();
END_METHOD

METHOD Test_DriveNoMovement
VAR
	nCycleCount : INT;	
END_VAR
TEST('Starter no movement, CW/CCW missing');

fbStarter.stConfig.fVelocity := 10;
fbStarter.stConfig.fAcceleration := 1000;
fbStarter.stConfig.fDeceleration := 1000;

fbStarter.stControlData.MotorCW := FALSE;
fbStarter.stControlData.MotorCCW := FALSE;
fbStarter.stControlData.BrakeActuation := TRUE;

fExpectedReal := 0;
bExpectedBool := FALSE;

FOR nCycleCount := 0 TO 10 DO
    fbStarter();
END_FOR

fResultReal := fbStarter.fSpeed;
bResultBool := fbStarter.stStatusData.MotorON;

AssertEquals(Expected := fExpectedReal,
             Actual := fResultReal,
             Message := 'fSpeed is not correct');	
			 
AssertEquals(Expected := bExpectedBool,
             Actual := bResultBool,
             Message := 'Status is not correct');		
			 
TEST_FINISHED();
//######################################################
TEST('Starter no movement, Brake missing, CW');

fbStarter.stConfig.fVelocity := 10;
fbStarter.stConfig.fAcceleration := 1000;
fbStarter.stConfig.fDeceleration := 1000;

fbStarter.stControlData.MotorCW := TRUE;
fbStarter.stControlData.MotorCCW := FALSE;
fbStarter.stControlData.BrakeActuation := FALSE;

fExpectedReal := 0;
bExpectedBool := FALSE;

FOR nCycleCount := 0 TO 10 DO
    fbStarter();
END_FOR

fResultReal := fbStarter.fSpeed;
bResultBool := fbStarter.stStatusData.MotorON;

AssertEquals(Expected := fExpectedReal,
             Actual := fResultReal,
             Message := 'DataOut is not correct');	
			 
AssertEquals(Expected := bExpectedBool,
             Actual := bResultBool,
             Message := 'Status is not correct');				 
			 		 
TEST_FINISHED();

//######################################################
TEST('Starter no movement, Brake missing, CCW');

fbStarter.stConfig.fVelocity := 10;
fbStarter.stConfig.fAcceleration := 1000;
fbStarter.stConfig.fDeceleration := 1000;

fbStarter.stControlData.MotorCW := FALSE;
fbStarter.stControlData.MotorCCW := TRUE;
fbStarter.stControlData.BrakeActuation := FALSE;

fExpectedReal := 0;
bExpectedBool := FALSE;

FOR nCycleCount := 0 TO 10 DO
    fbStarter();
END_FOR

fResultReal := fbStarter.fSpeed;
bResultBool := fbStarter.stStatusData.MotorON;

AssertEquals(Expected := fExpectedReal,
             Actual := fResultReal,
             Message := 'DataOut is not correct');	
			 
AssertEquals(Expected := bExpectedBool,
             Actual := bResultBool,
             Message := 'Status is not correct');			 
			 
TEST_FINISHED();
//######################################################
TEST('Starter no movement, CW and CCW active');

fbStarter.stConfig.fVelocity := 10;
fbStarter.stConfig.fAcceleration := 1000;
fbStarter.stConfig.fDeceleration := 1000;

fbStarter.stControlData.MotorCW := TRUE;
fbStarter.stControlData.MotorCCW := TRUE;
fbStarter.stControlData.BrakeActuation := TRUE;

fExpectedReal := 0;
bExpectedBool := FALSE;

FOR nCycleCount := 0 TO 10 DO
    fbStarter();
END_FOR

fResultReal := fbStarter.fSpeed;
bResultBool := fbStarter.stStatusData.MotorON;

AssertEquals(Expected := fExpectedReal,
             Actual := fResultReal,
             Message := 'DataOut is not correct');	
			 
AssertEquals(Expected := bExpectedBool,
             Actual := bResultBool,
             Message := 'Status is not correct');
			 
TEST_FINISHED();
END_METHOD

METHOD Test_DriveRunningCcw
VAR
	nCycleCount : INT;
END_VAR
TEST('Starter is running counter clock wise with 0 speed');
fbStarter.stControlData.MotorCW := FALSE;
fbStarter.stControlData.MotorCCW := TRUE;
fbStarter.stControlData.BrakeActuation := TRUE;

fbStarter.stConfig.fVelocity := 0;
fbStarter.stConfig.fAcceleration := 1000;
fbStarter.stConfig.fDeceleration := 1000;

fExpectedReal := 0;
bExpectedBool := FALSE;

FOR nCycleCount := 0 TO 100 DO
    fbStarter();
END_FOR

fResultReal := fbStarter.fSpeed;
bResultBool := fbStarter.stStatusData.MotorON;

AssertEquals(Expected := fExpectedReal,
             Actual := fResultReal,
             Message := 'DataOut is not correct');	
			 
AssertEquals(Expected := bExpectedBool,
             Actual := bResultBool,
             Message := 'Status is not correct');	
			 
fExpectedDataOut := fbStarter.GetLinkControlData();			 
AssertEquals(Expected := fExpectedReal,
             Actual := fExpectedDataOut,
             Message := 'DataOut is not correct');	
			 		 
TEST_FINISHED();
//######################################################
TEST('Starter is running counter clock wise with -100 speed');
fbStarter.stControlData.MotorCW := FALSE;
fbStarter.stControlData.MotorCCW := TRUE;
fbStarter.stControlData.BrakeActuation := TRUE;

fbStarter.stConfig.fVelocity := 10;
fbStarter.stConfig.fAcceleration := 1000;
fbStarter.stConfig.fDeceleration := 1000;

fExpectedReal := -10;
bExpectedBool := TRUE;

FOR nCycleCount := 0 TO 100 DO
    fbStarter();
END_FOR

fResultReal := fbStarter.fSpeed;
bResultBool := fbStarter.stStatusData.MotorON;

AssertEquals(Expected := fExpectedReal,
             Actual := fResultReal,
             Message := 'DataOut is not correct');	
			 
AssertEquals(Expected := bExpectedBool,
             Actual := bResultBool,
             Message := 'Status is not correct');
			 
TEST_FINISHED();
END_METHOD

METHOD Test_DriveRunningCw
VAR
	nCycleCount : INT;
END_VAR
TEST('Starter is running clock wise with 0 speed');
fbStarter.stControlData.MotorCW := TRUE;
fbStarter.stControlData.MotorCCW := FALSE;
fbStarter.stControlData.BrakeActuation := TRUE;

fbStarter.stConfig.fVelocity := 0;
fbStarter.stConfig.fAcceleration := 1000;
fbStarter.stConfig.fDeceleration := 1000;

fExpectedReal := 0;
bExpectedBool := FALSE;

FOR nCycleCount := 0 TO 10 DO
    fbStarter();
END_FOR

fResultReal := fbStarter.fSpeed;

bResultBool := fbStarter.stStatusData.MotorON;

AssertEquals(Expected := fExpectedReal,
             Actual := fResultReal,
             Message := 'DataOut is not correct');	
			 
AssertEquals(Expected := bExpectedBool,
             Actual := bResultBool,
             Message := 'Status is not correct');	
			 
TEST_FINISHED();
//######################################################
TEST('Starter is running clock wise with 100 speed');

fbStarter.stConfig.fVelocity := 10;
fbStarter.stConfig.fAcceleration := 1000;
fbStarter.stConfig.fDeceleration := 1000;

fbStarter.stControlData.MotorCW := TRUE;
fbStarter.stControlData.MotorCCW := FALSE;
fbStarter.stControlData.BrakeActuation := TRUE;

fExpectedReal := 10;
bExpectedBool := TRUE;

FOR nCycleCount := 0 TO 10 DO
    fbStarter();
END_FOR

fResultReal := fbStarter.fSpeed;
bResultBool := fbStarter.stStatusData.MotorON;

AssertEquals(Expected := fExpectedReal,
             Actual := fResultReal,
             Message := 'DataOut is not correct');	
			 
AssertEquals(Expected := bExpectedBool,
             Actual := bResultBool,
             Message := 'Status is not correct'); 
			 
TEST_FINISHED();
END_METHOD

METHOD Test_GetControlData : BOOL
VAR
	stExpectedControlData 	: ST_StarterControlData;
	nExpectedControlData	: WORD;	
	stActualControlData 	: ST_StarterControlData;
	nActualControlData		: WORD;		
	fbStarter 				: FB_Starter;	
END_VAR
TEST('Get Control Data');

stExpectedControlData.BrakeActuation := TRUE;
stExpectedControlData.DisQuickStop := TRUE;

MEMCPY(ADR(nExpectedControlData), ADR(stExpectedControlData), 2);

fbStarter.GetControlData(stActualControlData, ADR(nExpectedControlData), FALSE);
MEMCPY(ADR(nActualControlData), ADR(stActualControlData), 2);

AssertEquals(Expected := nExpectedControlData,
             Actual := nActualControlData,
             Message := 'nControlData is not equal');
		
TEST_FINISHED();
END_METHOD

METHOD Test_GetControlDataSWAP : BOOL
VAR
	stExpectedControlData 		: ST_StarterControlData;
	nExpectedControlData		: WORD;	
	nExpectedControlDataSWAP	: WORD;
	stActualControlData 		: ST_StarterControlData;
	nActualControlData			: WORD;		
	fbStarter 					: FB_Starter;	
END_VAR
TEST('Get Control Data SWAP');

stExpectedControlData.BrakeActuation := TRUE;
stExpectedControlData.DisQuickStop := TRUE;

MEMCPY(ADR(nExpectedControlData), ADR(stExpectedControlData), 2);
nExpectedControlDataSWAP := HOST_TO_BE16(nExpectedControlData);

fbStarter.GetControlData(stActualControlData, ADR(nExpectedControlDataSWAP), TRUE);
MEMCPY(ADR(nActualControlData), ADR(stActualControlData), 2);

AssertEquals(Expected := nExpectedControlData,
             Actual := nActualControlData,
             Message := 'nControlData is not equal');
		
TEST_FINISHED();
END_METHOD

METHOD Test_SetStatusData : BOOL
VAR
	stExpectedStatusData 	: ST_StarterStatusData;
	nExpectedStatusData		: WORD;	
	stActualStatusData 		: ST_StarterStatusData;
	nActualStatusData		: WORD;		
	fbStarter 				: FB_Starter;	
END_VAR
TEST('Set Status Data');

stExpectedStatusData.Ready := TRUE;
stExpectedStatusData.Input1 := TRUE;
stExpectedStatusData.Input2 := TRUE;

MEMCPY(ADR(nExpectedStatusData), ADR(stExpectedStatusData), 2);

fbStarter.SetStatusData(stExpectedStatusData, ADR(nActualStatusData), FALSE);

AssertEquals(Expected := nExpectedStatusData,
             Actual := nActualStatusData,
             Message := 'nStatusData is not equal');
		
TEST_FINISHED();
END_METHOD

METHOD Test_SetStatusDataSWAP : BOOL
VAR
	stExpectedStatusData 	: ST_StarterStatusData;
	nExpectedStatusData		: WORD;	
	stActualStatusData 		: ST_StarterStatusData;
	nActualStatusData		: WORD;		
	fbStarter 				: FB_Starter;	
END_VAR
TEST('Set Status Data SWAP');

stExpectedStatusData.Ready := TRUE;
stExpectedStatusData.Input1 := TRUE;
stExpectedStatusData.Input2 := TRUE;

MEMCPY(ADR(nExpectedStatusData), ADR(stExpectedStatusData), 2);
nExpectedStatusData := HOST_TO_BE16(nExpectedStatusData);

fbStarter.SetStatusData(stExpectedStatusData, ADR(nActualStatusData), TRUE);

AssertEquals(Expected := nExpectedStatusData,
             Actual := nActualStatusData,
             Message := 'nStatusData is not equal');
		
TEST_FINISHED();
END_METHOD

END_FUNCTION_BLOCK

// Tests/Safety/FB_Euchner_MGB_Test
FUNCTION_BLOCK FB_Euchner_MGB_Test EXTENDS FB_TestSuite
VAR
	fbEuchnerMgb : FB_EuchnerMGB;
	nExpected : BYTE;
	nResult : BYTE;
	bExpected : BOOL;
	bResult : BOOL;
END_VAR

Test_Button1();
Test_Button2();
Test_Button3();
Test_Button4();

Test_Lamp1();
Test_Lamp2();
Test_Lamp3();
Test_Lamp4();

Test_DoorOpen();
Test_DoorClosed_NoLock();
Test_DoorClosed_Locked();

METHOD Test_Button1
VAR_INPUT
END_VAR
TEST('Button 1 not pressed');
fbEuchnerMgb.SetStatus(0);
fbEuchnerMgb();
bExpected := FALSE;
bResult := fbEuchnerMgb.bButton_1;

AssertEquals(Expected := bExpected,
             Actual := bResult,
             Message := 'Value is not correct');	
TEST_FINISHED();

TEST('Button 1 is pressed');	
fbEuchnerMgb.SetStatus(16);
fbEuchnerMgb();
bExpected := TRUE;
bResult := fbEuchnerMgb.bButton_1;
AssertEquals(Expected := bExpected,
             Actual := bResult,
             Message := 'Control value is not correct');	 
TEST_FINISHED();
END_METHOD

METHOD Test_Button2
VAR_INPUT
END_VAR
TEST('Button 2 not pressed');
fbEuchnerMgb.SetStatus(0);
fbEuchnerMgb();
bExpected := FALSE;
bResult := fbEuchnerMgb.bButton_2;

AssertEquals(Expected := bExpected,
             Actual := bResult,
             Message := 'Value is not correct');	
TEST_FINISHED();

TEST('Button 2 is pressed');	
fbEuchnerMgb.SetStatus(32);
fbEuchnerMgb();
bExpected := TRUE;
bResult := fbEuchnerMgb.bButton_2;
AssertEquals(Expected := bExpected,
             Actual := bResult,
             Message := 'Control value is not correct');	 
TEST_FINISHED();
END_METHOD

METHOD Test_Button3
VAR_INPUT
END_VAR
TEST('Button 3 not pressed');
fbEuchnerMgb.SetStatus(0);
fbEuchnerMgb();
bExpected := FALSE;
bResult := fbEuchnerMgb.bButton_3;

AssertEquals(Expected := bExpected,
             Actual := bResult,
             Message := 'Value is not correct');	
TEST_FINISHED();

TEST('Button 3 is pressed');	
fbEuchnerMgb.SetStatus(64);
fbEuchnerMgb();
bExpected := TRUE;
bResult := fbEuchnerMgb.bButton_3;
AssertEquals(Expected := bExpected,
             Actual := bResult,
             Message := 'Control value is not correct');	 
TEST_FINISHED();
END_METHOD

METHOD Test_Button4
VAR_INPUT
END_VAR
TEST('Button 4 not pressed');
fbEuchnerMgb.SetStatus(0);
fbEuchnerMgb();
bExpected := FALSE;
bResult := fbEuchnerMgb.bButton_4;

AssertEquals(Expected := bExpected,
             Actual := bResult,
             Message := 'Value is not correct');	
TEST_FINISHED();

TEST('Button 4 is pressed');	
fbEuchnerMgb.SetStatus(128);
fbEuchnerMgb();
bExpected := TRUE;
bResult := fbEuchnerMgb.bButton_4;
AssertEquals(Expected := bExpected,
             Actual := bResult,
             Message := 'Control value is not correct');	 
TEST_FINISHED();
END_METHOD

METHOD Test_DoorClosed_Locked
VAR_INPUT
END_VAR
TEST('Door closed and locked');
fbEuchnerMgb.SetStatus(3);
fbEuchnerMgb.bLock := TRUE;
fbEuchnerMgb();
bExpected := TRUE;
bResult := fbEuchnerMgb.bclosed AND fbEuchnerMgb.bClosedAndLocked;

AssertEquals(Expected := bExpected,
             Actual := bResult,
             Message := 'Value is not correct');	
TEST_FINISHED();
END_METHOD

METHOD Test_DoorClosed_NoLock
VAR_INPUT
END_VAR
TEST('Door is closed but not locked');
fbEuchnerMgb.SetStatus(1);
fbEuchnerMgb();
bExpected := TRUE;
bResult := fbEuchnerMgb.bclosed AND NOT fbEuchnerMgb.bClosedAndLocked;

AssertEquals(Expected := bExpected,
             Actual := bResult,
             Message := 'Value is not correct');	
TEST_FINISHED();
END_METHOD

METHOD Test_DoorOpen
VAR_INPUT
END_VAR
TEST('Door is open');
fbEuchnerMgb.SetStatus(0);
fbEuchnerMgb();
bExpected := FALSE;
bResult := fbEuchnerMgb.bclosed;

AssertEquals(Expected := bExpected,
             Actual := bResult,
             Message := 'Value is not correct');	
TEST_FINISHED();
END_METHOD

METHOD Test_Lamp1
VAR_INPUT
END_VAR

VAR
	fbButton: INT;
END_VAR
TEST('Turn ON Lamp 1');			 
fbEuchnerMgb.bLamp_1 := TRUE; 
fbEuchnerMgb();
nExpected := 16;
nResult := fbEuchnerMgb.GetControl();
AssertEquals(Expected := nExpected,
             Actual := nResult,
             Message := 'Control value is not correct');	 
TEST_FINISHED();

TEST('Turn OFF Lamp 1');			 
fbEuchnerMgb.bLamp_1 := FALSE; 
fbEuchnerMgb();
nExpected := 0;
nResult := fbEuchnerMgb.GetControl();
AssertEquals(Expected := nExpected,
             Actual := nResult,
             Message := 'Control value is not correct');	 
TEST_FINISHED();
END_METHOD

METHOD Test_Lamp2
VAR_INPUT
END_VAR
TEST('Turn ON Lamp 2');			 
fbEuchnerMgb.bLamp_2 := TRUE; 
fbEuchnerMgb();
nExpected := 32;
nResult := fbEuchnerMgb.GetControl();
AssertEquals(Expected := nExpected,
             Actual := nResult,
             Message := 'Control value is not correct');	 
TEST_FINISHED();

TEST('Turn OFF Lamp 2');			 
fbEuchnerMgb.bLamp_2 := FALSE; 
fbEuchnerMgb();
nExpected := 0;
nResult := fbEuchnerMgb.GetControl();
AssertEquals(Expected := nExpected,
             Actual := nResult,
             Message := 'Control value is not correct');	 
TEST_FINISHED();
END_METHOD

METHOD Test_Lamp3
VAR_INPUT
END_VAR
TEST('Turn ON Lamp 3');			 
fbEuchnerMgb.bLamp_3 := TRUE; 
fbEuchnerMgb();
nExpected := 64;
nResult := fbEuchnerMgb.GetControl();
AssertEquals(Expected := nExpected,
             Actual := nResult,
             Message := 'Control value is not correct');	 
TEST_FINISHED();

TEST('Turn OFF Lamp 3');			 
fbEuchnerMgb.bLamp_3 := FALSE; 
fbEuchnerMgb();
nExpected := 0;
nResult := fbEuchnerMgb.GetControl();
AssertEquals(Expected := nExpected,
             Actual := nResult,
             Message := 'Control value is not correct');	 
TEST_FINISHED();
END_METHOD

METHOD Test_Lamp4
VAR_INPUT
END_VAR
TEST('Turn ON Lamp 4');			 
fbEuchnerMgb.bLamp_4 := TRUE; 
fbEuchnerMgb();
nExpected := 128;
nResult := fbEuchnerMgb.GetControl();
AssertEquals(Expected := nExpected,
             Actual := nResult,
             Message := 'Control value is not correct');	 
TEST_FINISHED();

TEST('Turn OFF Lamp 4');			 
fbEuchnerMgb.bLamp_4 := FALSE; 
fbEuchnerMgb();
nExpected := 0;
nResult := fbEuchnerMgb.GetControl();
AssertEquals(Expected := nExpected,
             Actual := nResult,
             Message := 'Control value is not correct');	 
TEST_FINISHED();
END_METHOD

END_FUNCTION_BLOCK

// Tests/Safety/FB_Euchner_STP_Test
FUNCTION_BLOCK FB_Euchner_STP_Test EXTENDS FB_TestSuite
VAR
	fbEuchnerStp : FB_EuchnerSTP;
	nExpected : BYTE;
	nResult : BYTE;
	bExpected : BOOL;
	bResult : BOOL;
END_VAR

Test_LampRD();
Test_LampGN();

Test_DoorOpen();
Test_DoorClosedAndUnlocked();
Test_DoorClosedAndLocked();

METHOD PRIVATE Test_DoorClosedAndLocked
VAR_INPUT
END_VAR
TEST('Door closed and locked');
fbEuchnerStp.SetStatus(3);
fbEuchnerStp.bLock := TRUE;
fbEuchnerStp();
bExpected := TRUE;
bResult := fbEuchnerStp.bclosed AND fbEuchnerStp.bClosedAndLocked;

AssertEquals(Expected := bExpected,
             Actual := bResult,
             Message := 'Value is not correct');	
TEST_FINISHED();
END_METHOD

METHOD PRIVATE Test_DoorClosedAndUnlocked
VAR_INPUT
END_VAR
TEST('Door is closed but not locked');
fbEuchnerStp.SetStatus(1);
fbEuchnerStp();
bExpected := TRUE;
bResult := fbEuchnerStp.bclosed AND NOT fbEuchnerStp.bClosedAndLocked;

AssertEquals(Expected := bExpected,
             Actual := bResult,
             Message := 'Value is not correct');	
TEST_FINISHED();
END_METHOD

METHOD PRIVATE Test_DoorOpen
VAR_INPUT
END_VAR
TEST('Door is open');
fbEuchnerStp.SetStatus(0);
fbEuchnerStp();
bExpected := FALSE;
bResult := fbEuchnerStp.bclosed;

AssertEquals(Expected := bExpected,
             Actual := bResult,
             Message := 'Value is not correct');	
TEST_FINISHED();
END_METHOD

METHOD PRIVATE Test_LampGN
VAR_INPUT
END_VAR
TEST('Turn ON Green lamp');			 
fbEuchnerStp.bLamp_GN := TRUE; 
fbEuchnerStp();
nExpected := 32;
nResult := fbEuchnerStp.GetControl();
AssertEquals(Expected := nExpected,
             Actual := nResult,
             Message := 'Control value is not correct');	 
TEST_FINISHED();

TEST('Turn OFF Green lamp');			 
fbEuchnerStp.bLamp_GN := FALSE; 
fbEuchnerStp();
nExpected := 0;
nResult := fbEuchnerStp.GetControl();
AssertEquals(Expected := nExpected,
             Actual := nResult,
             Message := 'Control value is not correct');	 
TEST_FINISHED();
END_METHOD

METHOD PRIVATE Test_LampRD
VAR_INPUT
END_VAR
TEST('Turn ON red lamp');			 
fbEuchnerStp.bLamp_RD := TRUE; 
fbEuchnerStp();
nExpected := 16;
nResult := fbEuchnerStp.GetControl();
AssertEquals(Expected := nExpected,
             Actual := nResult,
             Message := 'Control value is not correct');	 
TEST_FINISHED();

TEST('Turn OFF red lamp');			 
fbEuchnerStp.bLamp_RD := FALSE; 
fbEuchnerStp();
nExpected := 0;
nResult := fbEuchnerStp.GetControl();
AssertEquals(Expected := nExpected,
             Actual := nResult,
             Message := 'Control value is not correct');	 
TEST_FINISHED();
END_METHOD

END_FUNCTION_BLOCK

// Tests/PRG_TEST
PROGRAM PRG_TEST
VAR
	FB_System_Test : FB_System_Test;
	FB_Clamp01_Test : FB_Clamp01_Test;
	FB_Compare_Test : FB_Compare_Test;
	FB_Norm_Test : FB_Norm_Test;
	FB_Scale_Test : FB_Scale_Test;
	FB_Sign_Test : FB_Sign_Test;
	FB_InverBytesOrder_Test : FB_InverBytesOrder_Test;
	FB_GetByte_Test : FB_GetByte_Test;
	FB_Heater_Test : FB_Heater_Test;
	FB_MoveVelocity_Test : FB_MoveVelocity_Test;
	FB_MoveAbsolute_Test : FB_MoveAbsolute_Test; 
	FB_DriveControl_Test : FB_DriveControl_Test;
	FB_Button_Test : FB_Button_Test;
	FB_Switch_Test : FB_Switch_Test;
	FB_Lock_Test : FB_Lock_Test;
	FB_Panel_Test : FB_Panel_Test;
	FB_Cylinder_Test : FB_Cylinder_Test;
	FB_Device_Test : FB_Device_Test;
	FB_DeviceByte_Test : FB_DeviceByte_Test;
	FB_DeviceWord_Test : FB_DeviceWord_Test;
	FB_DeviceDWord_Test : FB_DeviceDWord_Test;
	FB_DeviceLWord_Test : FB_DeviceLWord_Test;
	FB_DeviceReal_Test : FB_DeviceReal_Test;
	FB_Drive_Test : FB_Drive_Test;
	FB_Lamp_Test : FB_Lamp_Test;
	FB_Reader_Test : FB_Reader_Test;
	FB_SensorAnalog_Test : FB_SensorAnalog_Test;
	FB_SensorBinary_Test : FB_SensorBinary_Test;
	FB_Robot_Test : FB_Robot_Test;
	FB_DS402FSM_Test : FB_DS402FSM_Test;
	FB_DS402_Test : FB_DS402_Test;
	FB_Euchner_MGB_Test : FB_Euchner_MGB_Test;
	FB_Euchner_STP_Test : FB_Euchner_STP_Test;
	FB_SimMovitracLTEB_Test : FB_SimMovitracLTEB_Test;
	FB_Starter_Test : FB_Starter_Test;
	FB_SimMovidriveFSM_Test : FB_SimMovidriveFSM_Test;
	FB_SimMovitrac_Test : FB_SimMovitrac_Test;
	FB_SimMovitracB_Test : FB_SimMovitracB_Test;
	FB_AdsMessageHandler_Test : FB_AdsMessageHandler_Test;
	FB_RecordData_Test : FB_RecordData_Test;
	FB_SimMovidrivePDO12_Test : FB_SimMovidrivePDO12_Test;
	FB_Encoder_Test : FB_Encoder_Test;
END_VAR

TcUnit.RUN();

END_PROGRAM

// Common/System/GVL_Core/fbSystem
PROPERTY PUBLIC fbSystem : REFERENCE TO FB_System
END_PROPERTY
